TYPE TransportComSubscribe :
STRUCT
  Request : TransportComRequest; // contains booleans that are used to start a specific sequence.
  Equipment : TransportComSubscribeEquipment;  // structs for equipment objects which are used by the bridges
END_STRUCT
END_TYPE

(* stored: Version 1.1.0.1
   DUT TransportComSubscribe: Id {561ca09a-4570-473d-a2c7-f1d68d4f0a46} *)
